(* PLC project Display.project, CODESYS V3.5 SP19 Patch 6 *)
(* stored: creationDateTime 2026-03-19T14:01:24.3469953+02:00, modificationDateTime 2026-03-19T14:01:24.3469953+02:00 *)

TYPE IdentityObject : STRUCT
  VendorId : DWORD := 0;  (* Vendor ID *)
  ProductCode : DWORD := 0;  (* Product code *)
  Revision : DWORD := 0;  (* Revision number *)
  SerialNumber : DWORD := 0;  (* Serial number for control unit *)
END_STRUCT;
END_TYPE

TYPE InitCanProtocolStates : (INIT_CANOPEN_PROTOCOLS := 1, INIT_CANOPEN_OD := 2, INIT_CANOPEN_PDO := 3, INIT_CANOPEN_OD_SAVE := 4, INIT_CANOPEN_OD_REORG := 5, INIT_CANOPEN_OD_REORG_READY := 6, INIT_INITIALIZE_OD_PARAMS := 7, INIT_INITIALIZE_OD_PARAMS_READY := 8, INIT_J1939 := 9, INIT_PROTOCOLS_DONE := 10);
END_TYPE

TYPE CAN1_TPDO_Bits : STRUCT
  Enable : BIT;  (* Bit[0] *)
  Set_BITS_Bit1 : BIT;  (* Bit[1] *)
  Set_BITS_Bit2 : BIT;  (* Bit[2] *)
  Set_BITS_Bit3 : BIT;  (* Bit[3] *)
  Set_BITS_Bit4 : BIT;  (* Bit[4] *)
  Set_BITS_Bit5 : BIT;  (* Bit[5] *)
  Set_BITS_Bit6 : BIT;  (* Bit[6] *)
  Set_BITS_Bit7 : BIT;  (* Bit[7] *)
END_STRUCT;
END_TYPE

TYPE CAN1_RPDO_RAU_Bits : STRUCT
  RAU_GPS_Init : BIT;  (* Bit[0] *)
  RAU_Bits_Bit1 : BIT;  (* Bit[1] *)
  RAU_Bits_Bit2 : BIT;  (* Bit[2] *)
  RAU_Bits_Bit3 : BIT;  (* Bit[3] *)
  RAU_Bits_Bit4 : BIT;  (* Bit[4] *)
  RAU_Bits_Bit5 : BIT;  (* Bit[5] *)
  RAU_Bits_Bit6 : BIT;  (* Bit[6] *)
  RAU_Bits_Bit7 : BIT;  (* Bit[7] *)
END_STRUCT;
END_TYPE

PROGRAM Main

                    
                      /// User code should be added to POU named as Main.
                    
                  
END_PROGRAM

PROGRAM MainInit
  VAR_OUTPUT
    o_MainInitReady : BOOL := FALSE;
  END_VAR

                    o_MainInitReady := TRUE;
                  
END_PROGRAM

(* Tool version : '8.6.9547.24640' (MultiTool build version) Xml version : '5.2' (MultiTool xml file version) Control Unit : 'Display' (Name of the unit in MultiTool) Control Unit Type : '6807' (Type of the unit in MultiTool, including the functional version) CODESYS Profile : 'CODESYS V3.5 SP19 Patch 6' (CODESYS profile that was selected in MultiTool) Device Description Version: '2.1.0.8' (Device description version that was selected in MultiTool) Export Time : '19.03.2026 14.01.24' (Date and time when exported from MultiTool) Export Path : 'C:\Codesys RPC\apps\CodesysRPC\Display' (Path where MultiTool exported) Project File : 'C:\Codesys RPC\apps\CodesysRPC\CodesysRPC.mtproject' (MultiTool project file name that was used) Libraries Path : 'C:\Codesys RPC\apps\CodesysRPC\Display\Libraries' *)
PROGRAM PLC_PRG

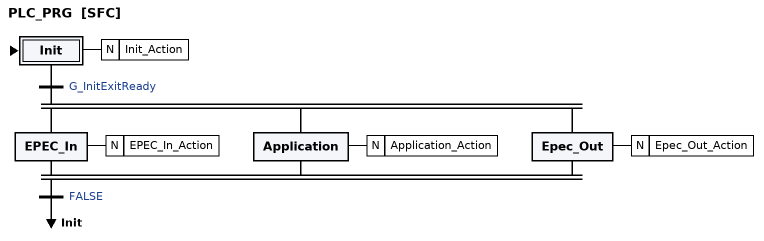
INITIAL_STEP Init:
  Init_Action(N);
END_STEP
TRANSITION FROM Init TO (EPEC_In, Application, Epec_Out)
  := G_InitExitReady;
END_TRANSITION
STEP EPEC_In:
  EPEC_In_Action(N);
END_STEP
TRANSITION FROM (EPEC_In, Application, Epec_Out) TO Init
  := FALSE;
END_TRANSITION
STEP Application:
  Application_Action(N);
END_STEP
STEP Epec_Out:
  Epec_Out_Action(N);
END_STEP

ACTION Application_Action:
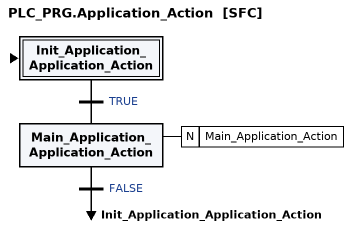
INITIAL_STEP Init_Application_Application_Action:
END_STEP
TRANSITION FROM Init_Application_Application_Action TO Main_Application_Application_Action
  := TRUE;
END_TRANSITION
STEP Main_Application_Application_Action:
  Main_Application_Action(N);
END_STEP
TRANSITION FROM Main_Application_Application_Action TO Init_Application_Application_Action
  := FALSE;
END_TRANSITION
END_ACTION

ACTION Bus_Action:
                        

G_CAN1_Channel.CheckMessages();
G_CAN2_Channel.CheckMessages();

(* Update callback data *)
IF G_CAN1_Channel.GetLatestError() <> DWORD#0 THEN
	G_CANopen_CAN1_VAR.Callback_Error := EPEC_CANopen.Errors.CallbackError;
ELSE
	G_CANopen_CAN1_VAR.Callback_Error := EPEC_CANopen.Errors.NoError;
END_IF

(* Update protocol data *)
G_CANopen_CAN1.HB_Handler.Update(
	i_Enable := TRUE,
	o_Error => G_CANopen_CAN1_VAR.HB_Error
);
G_CANopen_CAN1.NMT_Handler.Update(
	i_Enable := TRUE,
	o_Error => G_CANopen_CAN1_VAR.NMT_Error
);
G_CANopen_CAN1.SSDO_Handler.Update(
	i_Enable := TRUE,
	o_Error => G_CANopen_CAN1_VAR.SSDO_Error
);
G_CANopen_CAN1.GFC_Handler.Update(
	i_Enable := TRUE,
	o_Error => G_CANopen_CAN1_VAR.GFC_Error
);
G_CANopen_CAN1.PDO_Handler.Update(
	i_Enable := TRUE,
	o_Error => G_CANopen_CAN1_VAR.PDO_Error
);

G_CANopen_CAN1.OD_ReOrg.Update(o_Ready => , o_Error => G_CANopen_CAN1_VAR.OD_REORG_Error);

G_CANopen_CAN1.SaveODHandler.Update(i_Enable := TRUE,
	o_Ready => G_CANopen_CAN1_VAR.ODSave_OperationReady,
	o_Error => G_CANopen_CAN1_VAR.ODSave_Error);

IF G_CANopen_CAN1_VAR.HB_Error = EPEC_CANopen.Errors.NoError AND
	G_CANopen_CAN1_VAR.NMT_Error = EPEC_CANopen.Errors.NoError AND
	G_CANopen_CAN1_VAR.SSDO_Error = EPEC_CANopen.Errors.NoError AND
	G_CANopen_CAN1_VAR.GFC_Error = EPEC_CANopen.Errors.NoError AND
	G_CANopen_CAN1_VAR.PDO_Error = EPEC_CANopen.Errors.NoError AND
	G_CANopen_CAN1_VAR.OD_REORG_Error = EPEC_CANopen.Errors.NoError
THEN
	G_CANopenCan1ProtocolError := FALSE;
ELSE
	G_CANopenCan1ProtocolError := TRUE;
END_IF



(*Check for nmt reset *)
IF G_CANopen_CAN1.NMT.StateChanged THEN
	IF G_CANopen_CAN1.NMT.LastNmtCommand = EPEC_CANopen.NMTCommand.Reset OR 
	   G_CANopen_CAN1.NMT.LastNmtCommand = EPEC_CANopen.NMTCommand.ResetCommunication 
	THEN
		(* If there is NMT reset command for IEC application CANopen device,
			IEC application is started after IEC cycle in execution. *)
		G_RESET_MODULE := TRUE;
	END_IF
END_IF




                        
                      
END_ACTION

ACTION Diag_Action:
                        


(* HW diagnostic *)
    G_HWDiagnostics(
        i_SupplyVoltage  := WORD_TO_UINT(DEV_DSC_SUPPLY_Volt),
        i_SupplyVoltageHighLimit := G_SupplyVoltageHighLimit,
        i_SupplyVoltageLowLimit :=G_SupplyVoltageLowLimit,
        i_Ref5V := WORD_TO_UINT(DEV_DSC_REF_5V),
        i_Ref5VHighLimit :=  G_Ref5VHighLimit,
        i_Ref5VLowLimit := G_Ref5VLowLimit,
        i_PCBTemperature := DEV_DSC_TEMP_PCB,
        i_PCBTempHighLimit := G_TempPCBHighLimit,
        i_PCBTempLowLimit := G_TempPCBLowLimit,
        i_CPUTemperature := DEV_DSC_TEMP_CPU,
        i_CPUTempHighLimit := G_TempCPUHighLimit,
        i_CPUTempLowLimit := G_TempCPULowLimit,
        i_CycleTimeHighLimit := G_CycleTimeHighLimit,
        i_AIBiasVoltage	:= WORD_TO_UINT(DEV_DSC_AI_BIAS_Volt),
        i_RtcBackupVoltage := WORD_TO_UINT(DEV_DSC_RTC_BACKUP_Volt),
        i_Voltage12V := 0,
        i_AIBiasVoltageHighLimit := G_AIBiasVoltageHighLimit,
        i_AIBiasVoltageLowLimit := G_AIBiasVoltageLowLimit,
        i_RtcBackupVoltageLowLimit := G_RTCBackupVoltageLowLimit,
        i_Voltage12VHighLimit := 0,
        i_Voltage12VLowLimit := 0
    );

    SUPPLY_Volt := G_HWDiagnostics.o_SupplyVoltage;
    TEMP_PCB := G_HWDiagnostics.o_PCBTemperature;
    TEMP_CPU := G_HWDiagnostics.o_CPUTemperature;
    DEV_DSC_REF_OUT_5V_Enable := REF_OUT_5V_Enable;
    REF_OUT_5V_OK := (NOT DEV_DSC_REF_OUT_5V_ERROR) AND REF_OUT_5V_Enable;
	REF_5V := G_HWDiagnostics.o_Ref5V;
	AIBias_Volt := G_HWDiagnostics.o_AIBiasVoltage;
	RTCBackup_Volt := G_HWDiagnostics.o_RtcBackupVoltage;
	Voltage12V := G_HWDiagnostics.o_Voltage12V;
	ALS_Volt := DEV_DSC_ALS_Volt;

(* DO Sensing *)
	HWD_DOSensing_68xx(i_MeasuredVoltage := DEV_DSC_DO_DIAG_Volt);
	DEV_DSC_DO_DIAG_Enable := HWD_DOSensing_68xx.o_Enable;
	DEV_DSC_DO_DIAG_Selection := HWD_DOSensing_68xx.o_PinSelection;








(*########################################################*)
(*This block is created implicit. Don't add own code here.*)
(*########################################################*)

(* Diagnostics for CAN interfaces *)



(* CANopen networks management and diagnostics  *)



(* System Ok conditions *)
G_SystemOk:=NOT(G_HWDiagnostics.o_CPUTemperatureHigh) AND
		NOT(G_HWDiagnostics.o_CPUTemperatureLow) AND
		NOT(G_HWDiagnostics.o_PCBTemperatureHigh) AND
		NOT(G_HWDiagnostics.o_PCBTemperatureLow) AND
		NOT(G_HWDiagnostics.o_SupplyVoltageHigh) AND
		NOT(G_HWDiagnostics.o_SupplyVoltageLow) AND
		NOT(G_HWDiagnostics.o_CycleTimeHigh) AND
		NOT(G_HWDiagnostics.o_Ref5VHigh) AND
		NOT(G_HWDiagnostics.o_Ref5VLow) AND
		NOT(G_HWDiagnostics.o_AIBiasVoltageHigh) AND
		NOT(G_HWDiagnostics.o_AIBiasVoltageLow);

                        
                      
END_ACTION

ACTION EPEC_In_Action:
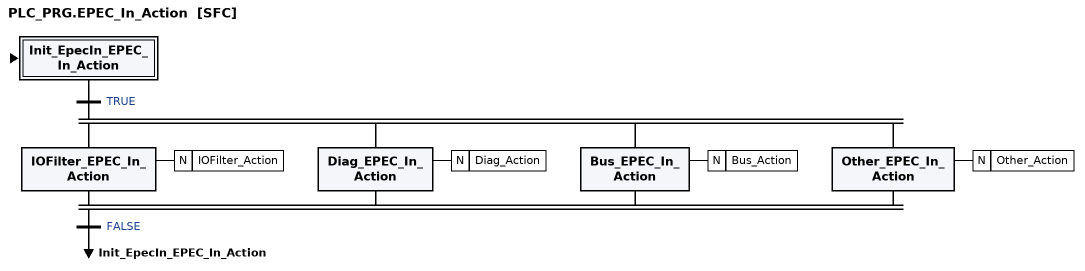
INITIAL_STEP Init_EpecIn_EPEC_In_Action:
END_STEP
TRANSITION FROM Init_EpecIn_EPEC_In_Action TO (IOFilter_EPEC_In_Action, Diag_EPEC_In_Action, Bus_EPEC_In_Action, Other_EPEC_In_Action)
  := TRUE;
END_TRANSITION
STEP IOFilter_EPEC_In_Action:
  IOFilter_Action(N);
END_STEP
TRANSITION FROM (IOFilter_EPEC_In_Action, Diag_EPEC_In_Action, Bus_EPEC_In_Action, Other_EPEC_In_Action) TO Init_EpecIn_EPEC_In_Action
  := FALSE;
END_TRANSITION
STEP Diag_EPEC_In_Action:
  Diag_Action(N);
END_STEP
STEP Bus_EPEC_In_Action:
  Bus_Action(N);
END_STEP
STEP Other_EPEC_In_Action:
  Other_Action(N);
END_STEP
END_ACTION

ACTION Epec_Out_Action:
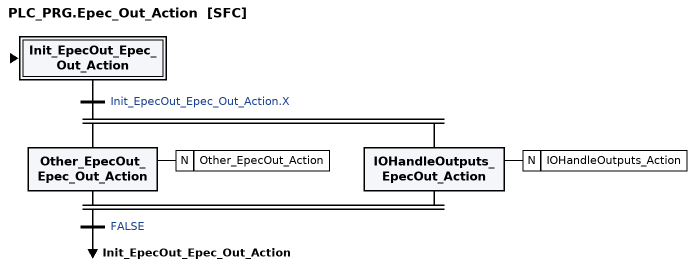
INITIAL_STEP Init_EpecOut_Epec_Out_Action:
END_STEP
TRANSITION FROM Init_EpecOut_Epec_Out_Action TO (Other_EpecOut_Epec_Out_Action, IOHandleOutputs_EpecOut_Action)
  := Init_EpecOut_Epec_Out_Action.X;
END_TRANSITION
STEP Other_EpecOut_Epec_Out_Action:
  Other_EpecOut_Action(N);
END_STEP
TRANSITION FROM (Other_EpecOut_Epec_Out_Action, IOHandleOutputs_EpecOut_Action) TO Init_EpecOut_Epec_Out_Action
  := FALSE;
END_TRANSITION
STEP IOHandleOutputs_EpecOut_Action:
  IOHandleOutputs_Action(N);
END_STEP
END_ACTION

ACTION Init_Action:
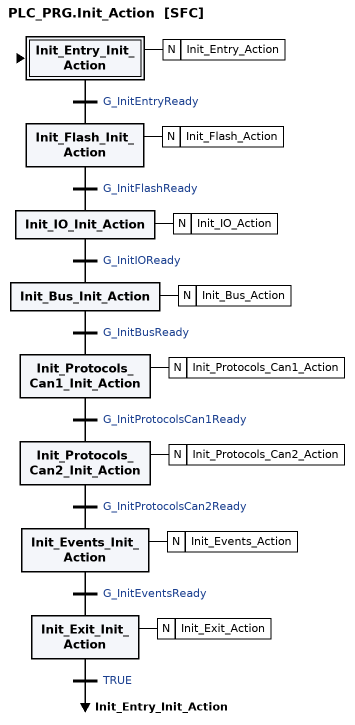
INITIAL_STEP Init_Entry_Init_Action:
  Init_Entry_Action(N);
END_STEP
TRANSITION FROM Init_Entry_Init_Action TO Init_Flash_Init_Action
  := G_InitEntryReady;
END_TRANSITION
STEP Init_Flash_Init_Action:
  Init_Flash_Action(N);
END_STEP
TRANSITION FROM Init_Flash_Init_Action TO Init_IO_Init_Action
  := G_InitFlashReady;
END_TRANSITION
STEP Init_IO_Init_Action:
  Init_IO_Action(N);
END_STEP
TRANSITION FROM Init_IO_Init_Action TO Init_Bus_Init_Action
  := G_InitIOReady;
END_TRANSITION
STEP Init_Bus_Init_Action:
  Init_Bus_Action(N);
END_STEP
TRANSITION FROM Init_Bus_Init_Action TO Init_Protocols_Can1_Init_Action
  := G_InitBusReady;
END_TRANSITION
STEP Init_Protocols_Can1_Init_Action:
  Init_Protocols_Can1_Action(N);
END_STEP
TRANSITION FROM Init_Protocols_Can1_Init_Action TO Init_Protocols_Can2_Init_Action
  := G_InitProtocolsCan1Ready;
END_TRANSITION
STEP Init_Protocols_Can2_Init_Action:
  Init_Protocols_Can2_Action(N);
END_STEP
TRANSITION FROM Init_Protocols_Can2_Init_Action TO Init_Events_Init_Action
  := G_InitProtocolsCan2Ready;
END_TRANSITION
STEP Init_Events_Init_Action:
  Init_Events_Action(N);
END_STEP
TRANSITION FROM Init_Events_Init_Action TO Init_Exit_Init_Action
  := G_InitEventsReady;
END_TRANSITION
STEP Init_Exit_Init_Action:
  Init_Exit_Action(N);
END_STEP
TRANSITION FROM Init_Exit_Init_Action TO Init_Entry_Init_Action
  := TRUE;
END_TRANSITION
END_ACTION

ACTION Init_Bus_Action:
                        (*###########################################################*)
(*This block is created implicit. Don't add own code to here.*)
(*###########################################################*)

G_CAN1_Channel.InitCAN(i_Channel:= EPEC_6000CANVXD.GVL_6000.CAN1, i_BitRate:=EPEC_CANVXD.BITRATE_250K, i_Flags:= 0);




G_InitBusReady := TRUE;

                        
                      
END_ACTION

ACTION Init_Entry_Action:
                        (*###########################################################*)
(*This block is created implicit. Don't add own code to here.*)
(*###########################################################*)

/// Call user init until flag is set on.
MainInit();
G_InitEntryReady := MainInit.o_MainInitReady;

IF TRUE = G_InitEntryReady THEN

EPEC_6000INT.GetUserFolder(i_pPath:=ADR(G_UserFolderPath),i_Length:=SIZEOF(G_UserFolderPath));


END_IF
                        
                      
END_ACTION

ACTION Init_Events_Action:
                        (*###########################################################*)
(*This block is created implicit. Don't add own code to here.*)
(*###########################################################*)
;



G_InitEventsReady:=TRUE;
                        
                      
END_ACTION

ACTION Init_Exit_Action:
                        (*###########################################################*)
(*This block is created implicit. Don't add own code to here.*)
(*###########################################################*)
;

G_NETWORK1_Parameters_CsvFile := Standard.CONCAT(STR1:=G_UserFolderPath, STR2:=G_NETWORK1_Parameters_CsvFile);
G_NETWORK1_Parameters_Count := EPEC_PAR.PARAMETERS_ReadCSV(i_Enable:=TRUE,
	i_File:=G_NETWORK1_Parameters_CsvFile,
	i_ParameterMaxCount:=G_NUMBER_OF_PARAMETERS_NETWORK1,
	i_pCSV:=0,
	i_itfExtraData:=0,
	o_CSVErrorCode=>G_NETWORK1_Parameters_ErrorCode,
	o_CSVErrorLine=>G_NETWORK1_Parameters_ErrorInLine);


G_UI.TimeSyncMethod := EPEC_6000INT.TimeSyncTypes.Manual;


G_InitExitReady:=TRUE;
                        
                      
END_ACTION

ACTION Init_Flash_Action:
                        (*###########################################################*)
(*This block is created implicit. Don't add own code to here.*)
(*###########################################################*)

G_InitFlashReady:=TRUE;
                        
                      
END_ACTION

ACTION Init_IO_Action:
                        (*###########################################################*)
(*This block is created implicit. Don't add own code to here.*)
(*###########################################################*)
;
(*IO init:*)
/// Init pin to AI mode Pin 1.5
DEV_DSC_AI_SET_mA_X1_5 := AI_SET_mA_X1_5;
DEV_DSC_AI_SET_PU_X1_5 := AI_SET_PU_X1_5;

/// Init pin to AI mode Pin 1.17
DEV_DSC_AI_SET_mA_X1_17 := AI_SET_mA_X1_17;
DEV_DSC_AI_SET_PU_X1_17 := AI_SET_PU_X1_17;


(*IO-init OK?*)
G_InitIOReady:=TRUE;
                        
                      
END_ACTION

ACTION Init_Protocols_Can1_Action:
                        (*###########################################################*)
(*This block is created implicit. Don't add own code to here.*)
(*###########################################################*)
;
CASE G_InitProtocolsCan1State OF

InitCanProtocolStates.INIT_CANOPEN_PROTOCOLS:
(*CAN1 INIT*)

G_CANopen_CAN1.Device.itfCanChannel:=G_CAN1_Channel; (*Connect device to can channel*)
G_CANopen_CAN1.Device.NodeID := BYTE#2;
G_CANopen_CAN1.NMT.NmtState:=EPEC_CANopen.NMTState.BootUp; (* Set NMT status to BOOTUP *)

(*Initialize OD's data structures*)
G_CANopen_CAN1.OD.EntryCount:=SIZEOF(G_CANopen_CAN1.ODEntrys)/SIZEOF(G_CANopen_CAN1.ODEntrys[1]); (*Max entries of given OD(CANopenDeviceODEntrys array)*)
G_CANopen_CAN1.OD.InOrder:=FALSE; (*OD isn't in order*)
G_CANopen_CAN1.OD.NextFree:=0; (*OD does not have any entries yet*)
G_CANopen_CAN1.OD.pODEntry:=ADR(G_CANopen_CAN1.ODEntrys); (*Pointer to OD array*)

(*Define NMT protocol*)
G_CANopen_CAN1.Protocols[1].Protocol:=EPEC_CANopen.ProtocolType.NMT;
G_CANopen_CAN1.Protocols[1].pData:=ADR(G_CANopen_CAN1.NMT);
G_CANopen_CAN1.Protocols[1].itfProtocol:=G_CANopen_CAN1.NMT_Handler;
G_CANopen_CAN1.Protocols[1].pError:=ADR(G_CANopen_CAN1_VAR.NMT_Error);
G_CANopen_CAN1_VAR.ProtocolAdded[1] := CANopenDeviceAddProtocol( (* Add to protocol stack *)
	i_pDevice:=ADR(G_CANopen_CAN1.Device),
	i_pProtocol:=ADR(G_CANopen_CAN1.Protocols[1]),
);

(*Initialize NMT protocol*)
IF G_CANopen_CAN1_VAR.ProtocolAdded[1] THEN
	G_CANopen_CAN1.NMT_Handler.Init(
		i_pDevice := ADR(G_CANopen_CAN1.Device),
		i_ThisIsMaster := TRUE,
		i_StartInterval :=  1000,
		i_pMonitoredNodes := ADR(G_CANopen_CAN1.MonitoredNodes),
		i_NumberOfNodes := 1,
		i_SimultaneousSlaveConfiguration := FALSE,
		i_pOdReOrg := ADR(G_CANopen_CAN1.OD_ReOrg),
		o_Error => G_CANopen_CAN1_VAR.NMT_Error
	);
ELSE
	G_CANopen_CAN1_VAR.NMT_Error := EPEC_CANopen.Errors.ProtocolDataMissing;
END_IF

(*Define OD protocol*)
G_CANopen_CAN1.Protocols[2].Protocol:=EPEC_CANopen.ProtocolType.OD;
G_CANopen_CAN1.Protocols[2].pData:=ADR(G_CANopen_CAN1.OD);
G_CANopen_CAN1.Protocols[2].pError:=ADR(G_CANopen_CAN1_VAR.OD_Error);
G_CANopen_CAN1_VAR.ProtocolAdded[2] := CANopenDeviceAddProtocol( (* Add to protocol stack *)
	i_pDevice:=ADR(G_CANopen_CAN1.Device),
	i_pProtocol:=ADR(G_CANopen_CAN1.Protocols[2]),
);
IF NOT G_CANopen_CAN1_VAR.ProtocolAdded[2] THEN
	G_CANopen_CAN1_VAR.OD_Error := EPEC_CANopen.Errors.ProtocolDataMissing;
END_IF

	(*Define HB protocol
	- Uses NMT and OD protocol data, thus need to be defined after them.
	*)
	G_CANopen_CAN1.HB.HeartBeat.PT := T#200MS; (* HB producer time *)
	G_CANopen_CAN1.HB.pHBCTimes := ADR(G_CANopen_CAN1_VAR.HBCTimes); (* HB consumer times *)

	G_CANopen_CAN1.Protocols[3].Protocol:=EPEC_CANopen.ProtocolType.HB;
	G_CANopen_CAN1.Protocols[3].pData:=ADR(G_CANopen_CAN1.HB);
	G_CANopen_CAN1.Protocols[3].itfProtocol:=G_CANopen_CAN1.HB_Handler;
	G_CANopen_CAN1.Protocols[3].pError:=ADR(G_CANopen_CAN1_VAR.HB_Error);
	G_CANopen_CAN1_VAR.ProtocolAdded[3] := CANopenDeviceAddProtocol( (* Add to protocol stack *)
		i_pDevice:=ADR(G_CANopen_CAN1.Device),
		i_pProtocol:=ADR(G_CANopen_CAN1.Protocols[3]),
	);

	(* Initialize HB protocol *)
	IF G_CANopen_CAN1_VAR.ProtocolAdded[3] THEN

		(* Add monitored nodes *)
		G_CANopen_CAN1.HB_Handler.AddCallbackToList(
			i_pDevice := ADR(G_CANopen_CAN1.Device),
			i_pCallback:=ADR(G_CANopen_CAN1.HBCallbacks[1]),
			o_Error => G_CANopen_CAN1_VAR.HB_Error
		);
		IF G_CANopen_CAN1_VAR.HB_Error = EPEC_CANopen.Errors.NoError THEN
			G_CANopen_CAN1.HB_Handler.Init(
				i_pDevice := ADR(G_CANopen_CAN1.Device),
				o_Error => G_CANopen_CAN1_VAR.HB_Error
			);
		END_IF
	ELSE
		G_CANopen_CAN1_VAR.HB_Error := EPEC_CANopen.Errors.ProtocolDataMissing;
	END_IF


(*Define SSDO protocol*)
G_CANopen_CAN1.Protocols[4].Protocol:=EPEC_CANopen.ProtocolType.SSDO;
G_CANopen_CAN1.Protocols[4].pData:=ADR(G_CANopen_CAN1.SSDO);
G_CANopen_CAN1.Protocols[4].itfProtocol:=G_CANopen_CAN1.SSDO_Handler;
G_CANopen_CAN1.Protocols[4].pError:=ADR(G_CANopen_CAN1_VAR.SSDO_Error);
G_CANopen_CAN1_VAR.ProtocolAdded[4] := CANopenDeviceAddProtocol( (* Add to protocol stack *)
	i_pDevice:=ADR(G_CANopen_CAN1.Device),
	i_pProtocol:=ADR(G_CANopen_CAN1.Protocols[4])
);
IF G_CANopen_CAN1_VAR.ProtocolAdded[4] THEN
	G_CANopen_CAN1.SSDO_Handler.Init(
		i_pDevice := ADR(G_CANopen_CAN1.Device),
		o_Error => G_CANopen_CAN1_VAR.SSDO_Error
	);
ELSE
	G_CANopen_CAN1_VAR.SSDO_Error := EPEC_CANopen.Errors.ProtocolDataMissing;
END_IF

(*Define PDO protocol*)
G_CANopen_CAN1.Protocols[5].Protocol:=EPEC_CANopen.ProtocolType.PDO;
G_CANopen_CAN1.Protocols[5].pData:=ADR(G_CANopen_CAN1.PDO);
G_CANopen_CAN1.Protocols[5].itfProtocol:=G_CANopen_CAN1.PDO_Handler;
G_CANopen_CAN1.Protocols[5].pError:=ADR(G_CANopen_CAN1_VAR.PDO_Error);
G_CANopen_CAN1_VAR.ProtocolAdded[5] := CANopenDeviceAddProtocol( (* Add to protocol stack *)
	i_pDevice:=ADR(G_CANopen_CAN1.Device),
	i_pProtocol:=ADR(G_CANopen_CAN1.Protocols[5])
);
IF G_CANopen_CAN1_VAR.ProtocolAdded[5] THEN
	G_CANopen_CAN1.PDO_Handler.Init(
		i_pDevice := ADR(G_CANopen_CAN1.Device),
		o_Error => G_CANopen_CAN1_VAR.PDO_Error
	);
ELSE
	G_CANopen_CAN1_VAR.PDO_Error := EPEC_CANopen.Errors.ProtocolDataMissing;
END_IF

(*Define GFC protocol*)
G_CANopen_CAN1.Protocols[6].Protocol:=EPEC_CANopen.ProtocolType.GFC;
G_CANopen_CAN1.Protocols[6].pData:=ADR(G_CANopen_CAN1.GFC);
G_CANopen_CAN1.Protocols[6].itfProtocol:=G_CANopen_CAN1.GFC_Handler;
G_CANopen_CAN1.Protocols[6].pError:=ADR(G_CANopen_CAN1_VAR.GFC_Error);
G_CANopen_CAN1_VAR.ProtocolAdded[6] := CANopenDeviceAddProtocol(  (* Add to protocol stack *)
	i_pDevice:=ADR(G_CANopen_CAN1.Device),
	i_pProtocol:=ADR(G_CANopen_CAN1.Protocols[6])
);
IF G_CANopen_CAN1_VAR.ProtocolAdded[6] THEN
	G_CANopen_CAN1.GFC_Handler.Init(
		i_pDevice := ADR(G_CANopen_CAN1.Device),
		i_pStatus:=ADR(G_CANopen_CAN1_VAR.GFC_Status),
		o_Error => G_CANopen_CAN1_VAR.GFC_Error
	);
ELSE
	G_CANopen_CAN1_VAR.GFC_Error := EPEC_CANopen.Errors.ProtocolDataMissing;
END_IF

(* Init CSDO instance array for bus *)
EPEC_CANopen.CANopenSDOManager.Init(
	i_pDevice:=ADR(G_CANopen_CAN1.Device),
	i_pCsdoArrayStart:=ADR(G_CANopen_CAN1.CSDOS),
	i_CsdoArraySize:=SIZEOF(G_CANopen_CAN1.CSDOS)/SIZEOF(G_CANopen_CAN1.CSDOS[1]),
	o_Error=>G_CANopen_CAN1_VAR.CSDO_Error
);





G_InitProtocolsCan1State := InitCanProtocolStates.INIT_CANOPEN_OD;

InitCanProtocolStates.INIT_CANOPEN_OD:

(*16#0001..16#0009 Default types *)
G_CANopen_CAN1_VAR.OD_Error := EPEC_CANopen.CANopenODAddDefautTypes(
	i_pOD:= ADR(G_CANopen_CAN1.OD)
);

	(* 16#1000 Information about the device type *)
	IF G_CANopen_CAN1_VAR.OD_Error = EPEC_CANopen.Errors.NoError THEN
		G_CANopen_CAN1_VAR.OD_Error := CANopenODAddLine(
			i_pOD := ADR(G_CANopen_CAN1.OD),(*Address of Object dictionary where index will be added*)
			i_Index := G_CANOPEN_ODINDEX_DEVICE_TYPE,
			i_ObjectCode := EPEC_CANopen.ObjectCode.OD_VAR,(*Type of index*)
			i_NumOfSubids := USINT#0,(*Number of subindexes*)
			i_TypeSpec := EPEC_CANopen.DataType.Deftype_UNSIGNED32,(*Index datatype, either user defined or standard CiA 301*)
			i_ObjectAccess := G_CANOPEN_OD_ACCESS_NOWRITE OR G_CANOPEN_OD_ACCESS_SUB0NOWRITE,
			i_Sub0data := USINT#0,(*Value of subindex0 in array or (def)struct*)
			i_pIndexData := ADR(G_CAN1_VAR.DeviceType_Device1),
			i_itfSDOHandler := DWORD#0
		);
	END_IF

	(* 16#1001 Error information *)
	IF G_CANopen_CAN1_VAR.OD_Error = EPEC_CANopen.Errors.NoError THEN
		G_CANopen_CAN1_VAR.OD_Error := CANopenODAddLine(
			i_pOD := ADR(G_CANopen_CAN1.OD),(*Address of Object dictionary where index will be added*)
			i_Index := G_CANOPEN_ODINDEX_ERROR_REGISTER,
			i_ObjectCode := EPEC_CANopen.ObjectCode.OD_VAR,(*Type of index*)
			i_NumOfSubids := USINT#0,(*Number of subindexes*)
			i_TypeSpec := EPEC_CANopen.DataType.Deftype_UNSIGNED8,(*Index datatype, either user defined or standard CiA 301*)
			i_ObjectAccess := G_CANOPEN_OD_ACCESS_NOWRITE OR G_CANOPEN_OD_ACCESS_SUB0NOWRITE,
			i_Sub0data := USINT#0,(*Value of subindex0 in array or (def)struct*)
			i_pIndexData := ADR(G_CAN1_VAR.ErrorReg_Device1),
			i_itfSDOHandler := DWORD#0
		);
	END_IF

	(* 16#1008 Manufacturer device name *)
	IF G_CANopen_CAN1_VAR.OD_Error = EPEC_CANopen.Errors.NoError THEN
		G_CANopen_CAN1_VAR.OD_Error := CANopenODAddLine(
			i_pOD := ADR(G_CANopen_CAN1.OD),(*Address of Object dictionary where index will be added*)
			i_Index := G_CANOPEN_ODINDEX_MF_DEVICE_NAME,
			i_ObjectCode := EPEC_CANopen.ObjectCode.OD_VAR,(*Type of index*)
			i_NumOfSubids := USINT#0,(*Number of subindexes*)
			i_TypeSpec := EPEC_CANopen.DataType.Deftype_STRING,(*Index datatype, either user defined or standard CiA 301*)
			i_ObjectAccess := G_CANOPEN_OD_ACCESS_NOWRITE OR G_CANOPEN_OD_ACCESS_SUB0NOWRITE,
			i_Sub0data := USINT#0,(*Value of subindex0 in array or (def)struct*)
			i_pIndexData := ADR(G_SystemInfo.DeviceName),
			i_itfSDOHandler := DWORD#0
		);
	END_IF

	(* 16#100A Manufacturer software version *)
	IF G_CANopen_CAN1_VAR.OD_Error = EPEC_CANopen.Errors.NoError THEN
		G_CANopen_CAN1_VAR.OD_Error := CANopenODAddLine(
			i_pOD := ADR(G_CANopen_CAN1.OD),(*Address of Object dictionary where index will be added*)
			i_Index := G_CANOPEN_ODINDEX_MF_SW_VERSION,
			i_ObjectCode := EPEC_CANopen.ObjectCode.OD_VAR,(*Type of index*)
			i_NumOfSubids := USINT#0,(*Number of subindexes*)
			i_TypeSpec := EPEC_CANopen.DataType.Deftype_STRING,(*Index datatype, either user defined or standard CiA 301*)
			i_ObjectAccess := G_CANOPEN_OD_ACCESS_NOWRITE OR G_CANOPEN_OD_ACCESS_SUB0NOWRITE,
			i_Sub0data := USINT#0,(*Value of subindex0 in array or (def)struct*)
			i_pIndexData := ADR(G_SystemInfo.SWVersion),
			i_itfSDOHandler := DWORD#0
		);
	END_IF

	(* 16#1018   Vendor ID *)
	IF G_CANopen_CAN1_VAR.OD_Error = EPEC_CANopen.Errors.NoError THEN
		G_CANopen_CAN1_VAR.OD_Error := CANopenODAddLine(
			i_pOD := ADR(G_CANopen_CAN1.OD),(*Address of Object dictionary where index will be added*)
			i_Index := G_CANOPEN_ODINDEX_IDENTITY_OBJECT,
			i_ObjectCode := EPEC_CANopen.ObjectCode.OD_ARRAY, (*Type of index*)
			i_NumOfSubids := USINT#4,(*Number of subindexes*)
			i_TypeSpec := EPEC_CANopen.DataType.Deftype_UNSIGNED32,(*Index of 16-bit deftype*)
			i_ObjectAccess := G_CANOPEN_OD_ACCESS_NOWRITE OR G_CANOPEN_OD_ACCESS_SUB0NOWRITE,
			i_Sub0data := USINT#4,(*Value of subindex0 in array or (def)struct*)
			i_pIndexData := ADR(G_SystemInfo.Identity),
			i_itfSDOHandler := DWORD#0
		);
	END_IF
	(* 16#2030   CodesysVersion *)
	IF G_CANopen_CAN1_VAR.OD_Error = EPEC_CANopen.Errors.NoError THEN
		G_CANopen_CAN1_VAR.OD_Error := CANopenODAddLine(
			i_pOD := ADR(G_CANopen_CAN1.OD),(*Address of Object dictionary where index will be added*)
			i_Index := 16#2030,
			i_ObjectCode := EPEC_CANopen.ObjectCode.OD_ARRAY, (*Type of index*)
			i_NumOfSubids := USINT#1,(*Number of subindexes*)
			i_TypeSpec := EPEC_CANopen.DataType.Deftype_UNSIGNED32,(*Index of 16-bit deftype*)
			i_ObjectAccess := G_CANOPEN_OD_ACCESS_READWRITE OR G_CANOPEN_OD_ACCESS_SUB0NOWRITE,
			i_Sub0data := USINT#1,(*Value of subindex0 in array or (def)struct*)
			i_pIndexData := ADR(G_SystemInfo.ToolsVersion),
			i_itfSDOHandler := DWORD#0
		);
	END_IF

	(* 16#2128 PDO Dummy Variable Index *)
	IF G_CANopen_CAN1_VAR.OD_Error = EPEC_CANopen.Errors.NoError THEN
		G_CANopen_CAN1_VAR.OD_Error := CANopenODAddLine(
			i_pOD := ADR(G_CANopen_CAN1.OD),(*Address of Object dictionary where index will be added*)
			i_Index := 16#2128,
			i_ObjectCode := EPEC_CANopen.ObjectCode.OD_VAR,(*Type of index*)
			i_NumOfSubids := USINT#0,(*Number of subindexes*)
			i_TypeSpec := EPEC_CANopen.DataType.Deftype_UNSIGNED8,(*Index datatype, either user defined or standard CiA 301*)
			i_ObjectAccess := G_CANOPEN_OD_ACCESS_READWRITE,
			i_Sub0data := USINT#0,(*Value of subindex0 in array or (def)struct*)
			i_pIndexData := ADR(G_CAN1_VAR.CAN1_TPDO_DUMMY),
			i_itfSDOHandler := DWORD#0
		);
	END_IF

	(* 16#2129 PDO Dummy Variable Index *)
	IF G_CANopen_CAN1_VAR.OD_Error = EPEC_CANopen.Errors.NoError THEN
		G_CANopen_CAN1_VAR.OD_Error := CANopenODAddLine(
			i_pOD := ADR(G_CANopen_CAN1.OD),(*Address of Object dictionary where index will be added*)
			i_Index := 16#2129,
			i_ObjectCode := EPEC_CANopen.ObjectCode.OD_VAR,(*Type of index*)
			i_NumOfSubids := USINT#0,(*Number of subindexes*)
			i_TypeSpec := EPEC_CANopen.DataType.Deftype_UNSIGNED8,(*Index datatype, either user defined or standard CiA 301*)
			i_ObjectAccess := G_CANOPEN_OD_ACCESS_READWRITE,
			i_Sub0data := USINT#0,(*Value of subindex0 in array or (def)struct*)
			i_pIndexData := ADR(G_CAN1_VAR.CAN1_RPDO_DUMMY),
			i_itfSDOHandler := DWORD#0
		);
	END_IF

	(* 16#2130   Application version *)
	IF G_CANopen_CAN1_VAR.OD_Error = EPEC_CANopen.Errors.NoError THEN
		G_CANopen_CAN1_VAR.OD_Error := CANopenODAddLine(
			i_pOD := ADR(G_CANopen_CAN1.OD),(*Address of Object dictionary where index will be added*)
			i_Index := 16#2130,
			i_ObjectCode := EPEC_CANopen.ObjectCode.OD_ARRAY, (*Type of index*)
			i_NumOfSubids := USINT#10,(*Number of subindexes*)
			i_TypeSpec := EPEC_CANopen.DataType.Deftype_STRING,(*Index of 16-bit deftype*)
			i_ObjectAccess := G_CANOPEN_OD_ACCESS_NOWRITE OR G_CANOPEN_OD_ACCESS_SUB0NOWRITE,
			i_Sub0data := USINT#10,(*Value of subindex0 in array or (def)struct*)
			i_pIndexData := ADR(G_SystemInfo.SoftwareInformation),
			i_itfSDOHandler := DWORD#0
		);
	END_IF

	(* 16#2131 Parameter CSV unique ID *)
	IF G_CANopen_CAN1_VAR.OD_Error = EPEC_CANopen.Errors.NoError THEN
		G_CANopen_CAN1_VAR.OD_Error := CANopenODAddLine(
			i_pOD := ADR(G_CANopen_CAN1.OD),(*Address of Object dictionary where index will be added*)
			i_Index := 16#2131,
			i_ObjectCode := EPEC_CANopen.ObjectCode.OD_VAR,(*Type of index*)
			i_NumOfSubids := USINT#0,(*Number of subindexes*)
			i_TypeSpec := EPEC_CANopen.DataType.Deftype_UNSIGNED16,(*Index datatype, either user defined or standard CiA 301*)
			i_ObjectAccess := G_CANOPEN_OD_ACCESS_NOWRITE OR G_CANOPEN_OD_ACCESS_SUB0NOWRITE,
			i_Sub0data := USINT#0,(*Value of subindex0 in array or (def)struct*)
			i_pIndexData := ADR(G_CAN1_VAR.Parameter_CSV_unique_ID1),
			i_itfSDOHandler := DWORD#0
		);
	END_IF

	(* 16#2140   MAC address byte 1 *)
	IF G_CANopen_CAN1_VAR.OD_Error = EPEC_CANopen.Errors.NoError THEN
		G_CANopen_CAN1_VAR.OD_Error := CANopenODAddLine(
			i_pOD := ADR(G_CANopen_CAN1.OD),(*Address of Object dictionary where index will be added*)
			i_Index := 16#2140,
			i_ObjectCode := EPEC_CANopen.ObjectCode.OD_ARRAY, (*Type of index*)
			i_NumOfSubids := USINT#6,(*Number of subindexes*)
			i_TypeSpec := EPEC_CANopen.DataType.Deftype_UNSIGNED8,(*Index of 16-bit deftype*)
			i_ObjectAccess := G_CANOPEN_OD_ACCESS_NOWRITE OR G_CANOPEN_OD_ACCESS_SUB0NOWRITE,
			i_Sub0data := USINT#6,(*Value of subindex0 in array or (def)struct*)
			i_pIndexData := ADR(G_SystemInfo.MACAddress),
			i_itfSDOHandler := DWORD#0
		);
	END_IF

	(* 16#2141   Ethernet enabled/disabled *)
	IF G_CANopen_CAN1_VAR.OD_Error = EPEC_CANopen.Errors.NoError THEN
		G_CANopen_CAN1_VAR.OD_Error := CANopenODAddLine(
			i_pOD := ADR(G_CANopen_CAN1.OD),(*Address of Object dictionary where index will be added*)
			i_Index := 16#2141,
			i_ObjectCode := EPEC_CANopen.ObjectCode.OD_ARRAY, (*Type of index*)
			i_NumOfSubids := USINT#50,(*Number of subindexes*)
			i_TypeSpec := EPEC_CANopen.DataType.Deftype_UNSIGNED8,(*Index of 16-bit deftype*)
			i_ObjectAccess := G_CANOPEN_OD_ACCESS_READWRITE OR G_CANOPEN_OD_ACCESS_SUB0NOWRITE,
			i_Sub0data := USINT#50,(*Value of subindex0 in array or (def)struct*)
			i_pIndexData := ADR(G_SystemInfo.EthernetConfiguration),
			i_itfSDOHandler := DWORD#0
		);
	END_IF

	(* 16#2150   Codesys communication enabled *)
	IF G_CANopen_CAN1_VAR.OD_Error = EPEC_CANopen.Errors.NoError THEN
		G_CANopen_CAN1_VAR.OD_Error := CANopenODAddLine(
			i_pOD := ADR(G_CANopen_CAN1.OD),(*Address of Object dictionary where index will be added*)
			i_Index := 16#2150,
			i_ObjectCode := EPEC_CANopen.ObjectCode.OD_ARRAY, (*Type of index*)
			i_NumOfSubids := USINT#10,(*Number of subindexes*)
			i_TypeSpec := EPEC_CANopen.DataType.Deftype_UNSIGNED16,(*Index of 16-bit deftype*)
			i_ObjectAccess := G_CANOPEN_OD_ACCESS_READWRITE OR G_CANOPEN_OD_ACCESS_SUB0NOWRITE,
			i_Sub0data := USINT#10,(*Value of subindex0 in array or (def)struct*)
			i_pIndexData := ADR(G_SystemInfo.CAN1_Comms),
			i_itfSDOHandler := DWORD#0
		);
	END_IF

	(* 16#2151   Codesys communication enabled *)
	IF G_CANopen_CAN1_VAR.OD_Error = EPEC_CANopen.Errors.NoError THEN
		G_CANopen_CAN1_VAR.OD_Error := CANopenODAddLine(
			i_pOD := ADR(G_CANopen_CAN1.OD),(*Address of Object dictionary where index will be added*)
			i_Index := 16#2151,
			i_ObjectCode := EPEC_CANopen.ObjectCode.OD_ARRAY, (*Type of index*)
			i_NumOfSubids := USINT#10,(*Number of subindexes*)
			i_TypeSpec := EPEC_CANopen.DataType.Deftype_UNSIGNED16,(*Index of 16-bit deftype*)
			i_ObjectAccess := G_CANOPEN_OD_ACCESS_READWRITE OR G_CANOPEN_OD_ACCESS_SUB0NOWRITE,
			i_Sub0data := USINT#10,(*Value of subindex0 in array or (def)struct*)
			i_pIndexData := ADR(G_SystemInfo.CAN2_Comms),
			i_itfSDOHandler := DWORD#0
		);
	END_IF

	(* 16#21EE Authentication status for non-safety parameter editing *)
	IF G_CANopen_CAN1_VAR.OD_Error = EPEC_CANopen.Errors.NoError THEN
		G_CANopen_CAN1_VAR.OD_Error := CANopenODAddLine(
			i_pOD := ADR(G_CANopen_CAN1.OD),(*Address of Object dictionary where index will be added*)
			i_Index := 16#21EE,
			i_ObjectCode := EPEC_CANopen.ObjectCode.OD_VAR,(*Type of index*)
			i_NumOfSubids := USINT#0,(*Number of subindexes*)
			i_TypeSpec := EPEC_CANopen.DataType.Deftype_UNSIGNED8,(*Index datatype, either user defined or standard CiA 301*)
			i_ObjectAccess := G_CANOPEN_OD_ACCESS_NOWRITE OR G_CANOPEN_OD_ACCESS_SUB0NOWRITE,
			i_Sub0data := USINT#0,(*Value of subindex0 in array or (def)struct*)
			i_pIndexData := ADR(G_CAN1_VAR.NonSafetyParameterAuthenticationStatus),
			i_itfSDOHandler := DWORD#0
		);
	END_IF

	(* 16#21EF Non-safety parameter password *)
	IF G_CANopen_CAN1_VAR.OD_Error = EPEC_CANopen.Errors.NoError THEN
		G_CANopen_CAN1_VAR.OD_Error := CANopenODAddLine(
			i_pOD := ADR(G_CANopen_CAN1.OD),(*Address of Object dictionary where index will be added*)
			i_Index := 16#21EF,
			i_ObjectCode := EPEC_CANopen.ObjectCode.OD_VAR,(*Type of index*)
			i_NumOfSubids := USINT#0,(*Number of subindexes*)
			i_TypeSpec := EPEC_CANopen.DataType.Deftype_STRING,(*Index datatype, either user defined or standard CiA 301*)
			i_ObjectAccess := G_CANOPEN_OD_ACCESS_SUB0NOREAD OR G_CANOPEN_OD_ACCESS_NOREAD,
			i_Sub0data := USINT#0,(*Value of subindex0 in array or (def)struct*)
			i_pIndexData := ADR(G_CAN1_VAR.NonSafetyParameterPassword),
			i_itfSDOHandler := DWORD#0
		);
	END_IF

	(* 16#5FB7 Automatically created REAL variables *)
	IF G_CANopen_CAN1_VAR.OD_Error = EPEC_CANopen.Errors.NoError THEN
		G_CANopen_CAN1_VAR.OD_Error := CANopenODAddLine(
			i_pOD := ADR(G_CANopen_CAN1.OD),(*Address of Object dictionary where index will be added*)
			i_Index := 16#5FB7,
			i_ObjectCode := EPEC_CANopen.ObjectCode.OD_ARRAY,(*Type of index*)
			i_NumOfSubids := USINT#6,(*Number of subindexes*)
			i_TypeSpec := EPEC_CANopen.DataType.Deftype_REAL32,(*Index datatype, either user defined or standard CiA 301*)
			i_ObjectAccess := G_CANOPEN_OD_ACCESS_READWRITE OR G_CANOPEN_OD_ACCESS_SUB0NOWRITE OR G_CANOPEN_OD_ACCESS_PDOMAP,
			i_Sub0data := USINT#6,(*Value of subindex0 in array or (def)struct*)
			i_pIndexData := ADR(G_CAN1_RPDO.RAU_GPS_altitude),
			i_itfSDOHandler := DWORD#0
		);
	END_IF

	(* 16#5FD7 Automatically created DWORD variables *)
	IF G_CANopen_CAN1_VAR.OD_Error = EPEC_CANopen.Errors.NoError THEN
		G_CANopen_CAN1_VAR.OD_Error := CANopenODAddLine(
			i_pOD := ADR(G_CANopen_CAN1.OD),(*Address of Object dictionary where index will be added*)
			i_Index := 16#5FD7,
			i_ObjectCode := EPEC_CANopen.ObjectCode.OD_ARRAY,(*Type of index*)
			i_NumOfSubids := USINT#3,(*Number of subindexes*)
			i_TypeSpec := EPEC_CANopen.DataType.Deftype_UNSIGNED32,(*Index datatype, either user defined or standard CiA 301*)
			i_ObjectAccess := G_CANOPEN_OD_ACCESS_READWRITE OR G_CANOPEN_OD_ACCESS_SUB0NOWRITE OR G_CANOPEN_OD_ACCESS_PDOMAP,
			i_Sub0data := USINT#3,(*Value of subindex0 in array or (def)struct*)
			i_pIndexData := ADR(G_CAN1_TPDO.PT100),
			i_itfSDOHandler := DWORD#0
		);
	END_IF

	(* 16#5FFF Automatically created BYTE variables *)
	IF G_CANopen_CAN1_VAR.OD_Error = EPEC_CANopen.Errors.NoError THEN
		G_CANopen_CAN1_VAR.OD_Error := CANopenODAddLine(
			i_pOD := ADR(G_CANopen_CAN1.OD),(*Address of Object dictionary where index will be added*)
			i_Index := 16#5FFF,
			i_ObjectCode := EPEC_CANopen.ObjectCode.OD_ARRAY,(*Type of index*)
			i_NumOfSubids := USINT#2,(*Number of subindexes*)
			i_TypeSpec := EPEC_CANopen.DataType.Deftype_UNSIGNED8,(*Index datatype, either user defined or standard CiA 301*)
			i_ObjectAccess := G_CANOPEN_OD_ACCESS_READWRITE OR G_CANOPEN_OD_ACCESS_SUB0NOWRITE OR G_CANOPEN_OD_ACCESS_PDOMAP,
			i_Sub0data := USINT#2,(*Value of subindex0 in array or (def)struct*)
			i_pIndexData := ADR(G_CAN1_TPDO.Bits),
			i_itfSDOHandler := DWORD#0
		);
	END_IF



G_InitProtocolsCan1State := InitCanProtocolStates.INIT_CANOPEN_PDO;

InitCanProtocolStates.INIT_CANOPEN_PDO:

	(* Init PDOs *)
	(* TPDO1 *)
	IF G_CANopen_CAN1_VAR.PDO_Error = EPEC_CANopen.Errors.NoError THEN
		G_CANopen_CAN1.PDOS[1].Init(
			i_pDevice:= ADR(G_CANopen_CAN1.Device),
			i_PDONumber := WORD#1,
			i_PDOType := EPEC_CANopen.PDOType.TransmitPDO,
			i_COB_ID := G_CANopen_CAN1.Device.NodeID + 16#180,
			i_TransmissionType := 16#FF,
			i_InhibitTime := 100,
			i_EventTime := 300,
			i_Mapping := G_CANopen_CAN1_Mappings.PDO1_Mappings,
			i_Mappings := 1,
			o_Error => G_CANopen_CAN1_VAR.PDO_Error
			);
	END_IF

	(* TPDO2 *)
	IF G_CANopen_CAN1_VAR.PDO_Error = EPEC_CANopen.Errors.NoError THEN
		G_CANopen_CAN1.PDOS[2].Init(
			i_pDevice:= ADR(G_CANopen_CAN1.Device),
			i_PDONumber := WORD#2,
			i_PDOType := EPEC_CANopen.PDOType.TransmitPDO,
			i_COB_ID := G_CANopen_CAN1.Device.NodeID + 16#280,
			i_TransmissionType := 16#FF,
			i_InhibitTime := 100,
			i_EventTime := 300,
			i_Mapping := G_CANopen_CAN1_Mappings.PDO2_Mappings,
			i_Mappings := 2,
			o_Error => G_CANopen_CAN1_VAR.PDO_Error
			);
	END_IF

	(* RAU_TPDO1 *)
	IF G_CANopen_CAN1_VAR.PDO_Error = EPEC_CANopen.Errors.NoError THEN
		G_CANopen_CAN1.PDOS[3].Init(
			i_pDevice:= ADR(G_CANopen_CAN1.Device),
			i_PDONumber := WORD#1,
			i_PDOType := EPEC_CANopen.PDOType.ReceivePDO,
			i_COB_ID := 16#181,
			i_TransmissionType := 16#FF,
			i_InhibitTime := 100,
			i_EventTime := 0,
			i_Mapping := G_CANopen_CAN1_Mappings.PDO3_Mappings,
			i_Mappings := 2,
			o_Error => G_CANopen_CAN1_VAR.PDO_Error
		);
	END_IF

	(* RAU_TPDO2 *)
	IF G_CANopen_CAN1_VAR.PDO_Error = EPEC_CANopen.Errors.NoError THEN
		G_CANopen_CAN1.PDOS[4].Init(
			i_pDevice:= ADR(G_CANopen_CAN1.Device),
			i_PDONumber := WORD#2,
			i_PDOType := EPEC_CANopen.PDOType.ReceivePDO,
			i_COB_ID := 16#281,
			i_TransmissionType := 16#FF,
			i_InhibitTime := 100,
			i_EventTime := 0,
			i_Mapping := G_CANopen_CAN1_Mappings.PDO4_Mappings,
			i_Mappings := 2,
			o_Error => G_CANopen_CAN1_VAR.PDO_Error
		);
	END_IF

	(* RAU_TPDO3 *)
	IF G_CANopen_CAN1_VAR.PDO_Error = EPEC_CANopen.Errors.NoError THEN
		G_CANopen_CAN1.PDOS[5].Init(
			i_pDevice:= ADR(G_CANopen_CAN1.Device),
			i_PDONumber := WORD#3,
			i_PDOType := EPEC_CANopen.PDOType.ReceivePDO,
			i_COB_ID := 16#381,
			i_TransmissionType := 16#FF,
			i_InhibitTime := 100,
			i_EventTime := 0,
			i_Mapping := G_CANopen_CAN1_Mappings.PDO5_Mappings,
			i_Mappings := 2,
			o_Error => G_CANopen_CAN1_VAR.PDO_Error
		);
	END_IF

	(* RAU_TPDO4 *)
	IF G_CANopen_CAN1_VAR.PDO_Error = EPEC_CANopen.Errors.NoError THEN
		G_CANopen_CAN1.PDOS[6].Init(
			i_pDevice:= ADR(G_CANopen_CAN1.Device),
			i_PDONumber := WORD#4,
			i_PDOType := EPEC_CANopen.PDOType.ReceivePDO,
			i_COB_ID := 16#481,
			i_TransmissionType := 16#FF,
			i_InhibitTime := 100,
			i_EventTime := 0,
			i_Mapping := G_CANopen_CAN1_Mappings.PDO6_Mappings,
			i_Mappings := 2,
			o_Error => G_CANopen_CAN1_VAR.PDO_Error
		);
	END_IF

	IF G_CANopen_CAN1_VAR.PDO_Error = EPEC_CANopen.Errors.NoError THEN
		G_CANopen_CAN1.PDO.pPDO:=ADR(G_CANopen_CAN1.PDOS);
		G_CANopen_CAN1.PDO.Count:=6; (* Amount of PDOS *)
	END_IF



G_InitProtocolsCan1State := InitCanProtocolStates.INIT_CANOPEN_OD_SAVE;

InitCanProtocolStates.INIT_CANOPEN_OD_SAVE:

(*Initialize OD save*)
G_CANopen_CAN1.SaveSubData1010h.pSaveSigns := ADR(G_CANopen_CAN1_VAR.SaveSigns1010[0]);
G_CANopen_CAN1.SaveSubData1010h.NumOfEntrys := 4;
G_CANopen_CAN1.SaveSubData1010h.pSaveIndexData := ADR(G_CANopen_CAN1.SaveData[0]);
G_CANopen_CAN1.SaveData[3].itfSaveAll := G_CANopen_CAN1.SaveAll;
G_CANopen_CAN1.SaveData[3].itfDeleteAll := G_CANopen_CAN1.DeleteAll;
G_CANopen_CAN1.OD.pAdditionalData := ADR(G_CANopen_CAN1.SaveSubData1010h);

IF G_CANopen_CAN1_VAR.OD_Error = EPEC_CANopen.Errors.NoError THEN
	G_CANopen_CAN1.SaveODHandler.Init(
		i_pOD:=ADR(G_CANopen_CAN1.OD),
		i_pSaveAll:= ADR(G_CANopen_CAN1.SaveAll),
		i_pDeleteAll:= ADR(G_CANopen_CAN1.DeleteAll),
		i_pParamHandler:=ADR(G_Common.ParHandler),
		i_NumOfParamsPerCycle:= 50,
		o_Error => G_CANopen_CAN1_VAR.ODSave_Error);
END_IF

G_CANopen_CAN1.OD_ReOrg.Init(i_pOD := ADR(G_CANopen_CAN1.OD), i_NumOfODIndexPerCycle := 50);
G_CANopen_CAN1.OD_ReOrg.Start();

G_InitProtocolsCan1State := InitCanProtocolStates.INIT_CANOPEN_OD_REORG;

InitCanProtocolStates.INIT_CANOPEN_OD_REORG:

G_CANopen_CAN1.OD_ReOrg.Update(o_Ready => G_CANopen_CAN1_VAR.OdReOrgReady, o_Error => G_CANopen_CAN1_VAR.OD_REORG_Error);

IF G_CANopen_CAN1_VAR.OdReOrgReady THEN
	(* Check all protocol init status flags *)
	IF G_CANopen_CAN1_VAR.NMT_Error = EPEC_CANopen.Errors.NoError AND
		G_CANopen_CAN1_VAR.SSDO_Error = EPEC_CANopen.Errors.NoError AND
		G_CANopen_CAN1_VAR.OD_Error = EPEC_CANopen.Errors.NoError AND
		G_CANopen_CAN1_VAR.HB_Error = EPEC_CANopen.Errors.NoError AND
		G_CANopen_CAN1_VAR.CSDO_Error = EPEC_CANopen.Errors.NoError AND
		G_CANopen_CAN1_VAR.GFC_Error = EPEC_CANopen.Errors.NoError AND
		G_CANopen_CAN1_VAR.PDO_Error = EPEC_CANopen.Errors.NoError AND
		G_CANopen_CAN1_VAR.OD_REORG_Error = EPEC_CANopen.Errors.NoError
	THEN
		G_InitCANopenCan1Error := FALSE; (* No errors in protocol inits *)
	ELSE
		G_InitCANopenCan1Error := TRUE;
	END_IF
	G_InitProtocolsCan1State := InitCanProtocolStates.INIT_CANOPEN_OD_REORG_READY;
END_IF

InitCanProtocolStates.INIT_CANOPEN_OD_REORG_READY:
	G_InitProtocolsCan1State := INIT_INITIALIZE_OD_PARAMS;

INIT_INITIALIZE_OD_PARAMS:
	G_CANopen_CAN1.SaveODHandler.InitializeODParams(i_Enable:=TRUE,
		o_Ready=>G_CANopen_CAN1_VAR.ODParametersInitialized,
		o_Error=>G_CANopen_CAN1_VAR.ODSave_Error);

	IF G_CANopen_CAN1_VAR.ODParametersInitialized THEN
		G_InitProtocolsCan1State := InitCanProtocolStates.INIT_INITIALIZE_OD_PARAMS_READY;
	END_IF

INIT_INITIALIZE_OD_PARAMS_READY:


G_InitProtocolsCan1State := InitCanProtocolStates.INIT_J1939;

InitCanProtocolStates.INIT_J1939:



G_InitProtocolsCan1State := InitCanProtocolStates.INIT_PROTOCOLS_DONE;

InitCanProtocolStates.INIT_PROTOCOLS_DONE:
G_InitProtocolsCan1Ready := TRUE;

END_CASE
                        
                      
END_ACTION

ACTION Init_Protocols_Can2_Action:
                        (*###########################################################*)
(*This block is created implicit. Don't add own code to here.*)
(*###########################################################*)
;
CASE G_InitProtocolsCan2State OF

InitCanProtocolStates.INIT_CANOPEN_PROTOCOLS:
(*CAN2 INIT*)





G_InitProtocolsCan2State := InitCanProtocolStates.INIT_CANOPEN_OD;

InitCanProtocolStates.INIT_CANOPEN_OD:



G_InitProtocolsCan2State := InitCanProtocolStates.INIT_CANOPEN_PDO;

InitCanProtocolStates.INIT_CANOPEN_PDO:



G_InitProtocolsCan2State := InitCanProtocolStates.INIT_CANOPEN_OD_SAVE;

InitCanProtocolStates.INIT_CANOPEN_OD_SAVE:



G_InitProtocolsCan2State := InitCanProtocolStates.INIT_J1939;

InitCanProtocolStates.INIT_J1939:



G_InitProtocolsCan2State := InitCanProtocolStates.INIT_PROTOCOLS_DONE;

InitCanProtocolStates.INIT_PROTOCOLS_DONE:
G_InitProtocolsCan2Ready := TRUE;

END_CASE
                        
                      
END_ACTION

ACTION IOFilter_Action:
                        ;

/// Handle AI channel Pin 1.5
DEV_DSC_AI_SET_mA_X1_5 := AI_SET_mA_X1_5;
DEV_DSC_AI_SET_PU_X1_5 := AI_SET_PU_X1_5;
AI_X1_5 := DEV_DSC_AI_RAW_X1_5;
AI_PU_X1_5 := DEV_DSC_AI_PU_X1_5;


/// KL15 Pin 1.6
KL15_X1_6 := DEV_DSC_KL15;



/// Handle AI channel Pin 1.17
DEV_DSC_AI_SET_mA_X1_17 := AI_SET_mA_X1_17;
DEV_DSC_AI_SET_PU_X1_17 := AI_SET_PU_X1_17;
AI_X1_17 := DEV_DSC_AI_RAW_X1_17;
AI_PU_X1_17 := DEV_DSC_AI_PU_X1_17;


                        
                      
END_ACTION

ACTION IOHandleOutputs_Action:
                        ;
DEV_DSC_BUZZER := BUZZER_CONTROL;

                        
                      
END_ACTION

ACTION Main_Application_Action:
                        (* Call user application *)
Main();
                        
                      
END_ACTION

ACTION Other_Action:
                        (*###########################################################*)
(*This block is created implicit. Don't add own code to here.*)
(*###########################################################*)


                        
                      
END_ACTION

ACTION Other_EpecOut_Action:
                        (* tag EPEC_OUT_OTHER *)


IF G_Common.ParHandler.o_ParamAreaLocked THEN
	G_Common.ParHandler.DisableChanges(i_DisableChanges := FALSE);
END_IF


                      
END_ACTION
END_PROGRAM

CONFIGURATION Device
  RESOURCE Application ON PLC
    VAR_GLOBAL CONSTANT  (* Code_Template_constants *)
      G_NVRAM_6107_CODE_TEMPLATE_TOTAL : DWORD := 507904;  (* [Total size of NVRAM reserved for code template (IEC area 496 kB)] *)
      G_NVRAM_6107_GLOBE_DATA_SIZE : DWORD := 1024;  (* [Size of the GlobE NVRAM reservation] *)
      G_NVRAM_6107_AZURE_DATA_SIZE : DWORD := 1024;  (* [Size of the Azure NVRAM reservation] *)
      G_NVRAM_6107_AZURE_DATA_OFFSET : DWORD := 490496;  (* [Offset of the Azure NVRAM area.] *)
      G_NVRAM_6107_GLOBE_DATA_OFFSET : DWORD := 491520;  (* [Offset of the GlobE NVRAM area.] *)
      G_NUMBER_OF_PARAMETERS_NETWORK1 : INT := 0;  (* [Number of parameters in network] *)
      G_NVRAM_6107_OD_PAR_IMAGE_SIZE : DWORD := 204800;  (* [Size of the OD parameter area reservation.] *)
      G_NVRAM_6107_EVENT_LOG_SIZE : DWORD := 102400;  (* [Size of the EventLog reservation.] *)
      G_NVRAM_6107_USER_DATA_SIZE : DWORD := 102400;  (* [Size of the user NVRAM reservation.] *)
      G_NVRAM_6107_OD_PARAM_OFFSET : DWORD := 0;  (* [Offset for OD parameter area.] *)
      G_NVRAM_6107_EVENTLOG_OFFSET : DWORD := 204800;  (* [Offset of the EventLog area.] *)
      G_NVRAM_6107_USER_DATA_OFFSET : DWORD := 307200;  (* [Offset of the user NVRAM area.] *)
      G_NVRAM_MACHINETYPE_OFFSET : DWORD := 409600;  (* [Offset of the machine type area.] *)
      G_PARAMHANDLERKEYWORD : DWORD := 16#2464842F;  (* [ Parameterhandler keyword] *)
      G_PARAM_BLOCK_MAX_SIZE : WORD := 1024;  (* [ Maximum size of one parameter handler block] *)
      G_NVRAM_MACHINETYPE_SIZE : DWORD := 0;  (* [Size of the machine type area reservation.] *)
    END_VAR
    VAR_GLOBAL  (* Code_Template_globals *)
      G_RESET_MODULE : BOOL := FALSE;  (* [Flag indicates if unit is wanted to reset after current application cycle. Reset actions can be varied between platforms.] *)
      G_HWDiagnostics : HWD_Measurements_68xx;  (* [Function block instance which is used for voltage and temperature monitoring.] *)
      G_AddAllAutoGenEventsToLog : BOOL := TRUE;  (* [Add all automatically generated events to log.] *)
      G_OffDelayForAutoGenEvents : WORD := 50;  (* [Off delay for automatically generated events.] *)
      G_OnDelayForAutoGenEvents : WORD := 100;  (* [On delay for automatically generated events.] *)
      G_AIOverCurrentProtection_X1_5 : EPEC_6000INT.AIOverCurrentProtection;
      G_AIOverCurrentProtectionEnable_X1_5 : BOOL := TRUE;
      G_AIOverCurrentProtection_X1_17 : EPEC_6000INT.AIOverCurrentProtection;
      G_AIOverCurrentProtectionEnable_X1_17 : BOOL := TRUE;
      G_SystemOk : BOOL := FALSE;
      G_TempCPUHighLimit : INT := 900;
      G_TempCPULowLimit : INT := -300;
      G_TempPCBHighLimit : INT := 900;
      G_TempPCBLowLimit : INT := -300;
      G_SupplyVoltageHighLimit : UINT := 3000;
      G_SupplyVoltageLowLimit : UINT := 0;
      G_CycleTimeHighLimit : UINT := 50;
      G_Ref5VHighLimit : UINT := 550;
      G_Ref5VLowLimit : UINT := 450;
      G_AIBiasVoltageHighLimit : UINT := 780;
      G_AIBiasVoltageLowLimit : UINT := 680;
      G_RtcBackupVoltageLowLimit : UINT := 200;
      G_NVRAM_6107_StartAddress : DWORD;  (* [Pointer to the start of the NVRAM area.] *)
      G_NVRAM_6107_ODParamPointer : DWORD;  (* [Pointer to the start of the OD parameter image.] *)
      G_NVRAM_6107_EventLogPointer : DWORD;  (* [Pointer to the start of the EventLog] *)
      G_NVRAM_6107_UserDataPointer : DWORD;  (* [Pointer to the start of the user NVRAM area.] *)
      G_NVRAM_6107_GlobEDataPointer : DWORD;  (* [Pointer to the start of the GlobE NVRAM area.] *)
      G_NVRAM_6107_AzureDataPointer : DWORD;  (* [Pointer to the start of the Azure NVRAM area.] *)
      G_NVRAM_6107_J1939DM2LogPointer : DWORD;  (* [Pointer to the start of the J1939 DM2 NVRAM area.] *)
      G_NVRAM_MachineTypePointer : DWORD;  (* [Pointer to the start of the Machine type NVRAM area.] *)
      G_InitEntryReady : BOOL := FALSE;  (* [Init Flags] *)
      G_InitFlashReady : BOOL := FALSE;
      G_InitIOReady : BOOL := FALSE;
      G_InitBusReady : BOOL := FALSE;
      G_InitProtocolsCan1Ready : BOOL := FALSE;
      G_InitProtocolsCan2Ready : BOOL := FALSE;
      G_InitEventsReady : BOOL := FALSE;
      G_InitExitReady : BOOL := FALSE;
      G_ActiveError : BOOL := FALSE;
      G_MRAM_Shm : SystemSharedMemRegion;  (* [Shared memory structure which is used to get pointer to MRAM area for parameter saving.] *)
      G_CommsParamCounterSaveCmdOld : WORD := 0;  (* [Counter used to detect if communication parameters need to be saved] *)
      G_CommsParamCounterRestoreCmdOld : WORD := 0;  (* [Counter used to detect if communication parameters need to be restored] *)
      G_NodeIds : ARRAY[1..2] OF INT := [2, 2];
      G_CAN1_Channel : EPEC_6000CANVXD.Channel;
      G_InitProtocolsCan1State : InitCanProtocolStates := INIT_CANOPEN_PROTOCOLS;
      G_InitCANopenCan1Error : BOOL := FALSE;
      G_CANopenCan1ProtocolError : BOOL := FALSE;
      G_CAN2_Channel : EPEC_6000CANVXD.Channel;
      G_InitProtocolsCan2State : InitCanProtocolStates := INIT_CANOPEN_PROTOCOLS;
      G_InitCANopenCan2Error : BOOL := FALSE;
      G_CANopenCan2ProtocolError : BOOL := FALSE;
      G_NETWORK1_Parameters_CSVData : ARRAY[1..G_NUMBER_OF_PARAMETERS_NETWORK1] OF EPEC_PAR.CSVData;  (* [Parameter CSV configuration parameters] *)
      G_NETWORK1_Parameters_CsvFile : STRING(79) := 'Parameters_NETWORK1.csv';  (* [CSV file path and name] *)
      G_NETWORK1_Parameters_Count : INT;  (* [CSV File parameter count] *)
      G_NETWORK1_Parameters_ErrorCode : EPEC_PAR.CSVError;  (* [CSV error code] *)
      G_NETWORK1_Parameters_ErrorInLine : INT;  (* [Number of CSV line containing error] *)
      G_UserFolderPath : STRING(255);
    END_VAR
    VAR_GLOBAL  (* UserMramVariables *)
      G_pUserMramStructure : POINTER TO UserMramStructure;  (* [Pointer to the start of the NVRAM area.] *)
      G_UserMramStructureDefault : UserMramStructure;  (* [Pointer to the start of the OD parameter image.] *)
    END_VAR
    VAR_GLOBAL  (* IO *)
      AI_PU_X1_5 : WORD := 0;  (* [Pin 1.5 - lang.IO.FilteredAiValue] *)
      AI_X1_5 : WORD := 0;  (* [Pin 1.5 - lang.IO.FilteredAiValue] *)
      KL15_X1_6 : BOOL := FALSE;  (* [Pin 1.6 - KL15] *)
      AI_PU_X1_17 : WORD := 0;  (* [Pin 1.17 - lang.IO.FilteredAiValue] *)
      AI_X1_17 : WORD := 0;  (* [Pin 1.17 - lang.IO.FilteredAiValue] *)
    END_VAR
    VAR_GLOBAL  (* IO_INTERNAL *)
      TEMP_PCB : INT := 0;  (* Scaled PCB temperature [0.1 C] *)
      TEMP_CPU : INT := 0;  (* Scaled CPU temperature [0.1 C] *)
      SUPPLY_Volt : WORD := 0;  (* Scaled supply voltage [0.01 V] *)
      AIBias_Volt : WORD := 0;  (* Scaled AI bias voltage *)
      RTCBackup_Volt : WORD := 0;  (* Scaled RTC backup voltage *)
      Voltage12V : WORD := 0;  (* Scaled 12V voltage *)
      REF_5V : WORD := 0;  (* Scaled Ref 5 V voltage [10 mV]. *)
      REF_OUT_5V_Enable : BOOL := FALSE;  (* Enable for 5 V reference. *)
      REF_OUT_5V_OK : BOOL := FALSE;  (* 5 V refrence failure *)
      BUZZER_CONTROL : BOOL := FALSE;  (* Enable buzzer output control *)
      ALS_Volt : WORD := 0;  (* Unscaled ALS voltage measurement *)
    END_VAR
    VAR_GLOBAL  (* IO_CONFIG *)
      AI_SET_PU_X1_5 : BOOL := TRUE;  (* [Pin 1.5 - lang.IO.PullUpEnableSelectionForPin] *)
      AI_SET_mA_X1_5 : BOOL := FALSE;  (* [Pin 1.5 - lang.IO.ModeSelection] *)
      AI_SET_PU_X1_17 : BOOL := TRUE;  (* [Pin 1.17 - lang.IO.PullUpEnableSelectionForPin] *)
      AI_SET_mA_X1_17 : BOOL := FALSE;  (* [Pin 1.17 - lang.IO.ModeSelection] *)
    END_VAR
    {attribute 'qualified_only'}
    {attribute 'location' := '16#800'}
    {attribute 'analysis' := '-5, -6, -33, -43, -48'}
    VAR_GLOBAL  (* G_CAN1_VAR - NOTE! NOTE! NOTE! NOTE! NOTE! NOTE! NOTE! NOTE! NOTE! NOTE! NOTE! This object is created by Epec MultiTool User changes are overwritten when project is imported Content - CANopen OD index data *)
      DeviceType_Device1 : UDINT := 405;  (* [ 16#1000 Information about the device type] *)
      ErrorReg_Device1 : USINT := 0;  (* [ 16#1001 Error information] *)
      CAN1_TPDO_DUMMY : BYTE := 0;  (* [ 16#2128 PDO Dummy Variable Index] *)
      CAN1_RPDO_DUMMY : BYTE := 0;  (* [ 16#2129 PDO Dummy Variable Index] *)
      Parameter_CSV_unique_ID1 : UINT := 16#0000;  (* [ 16#2131 Parameter CSV unique ID] *)
      NonSafetyParameterAuthenticationStatus : BYTE := 0;  (* [ 16#21EE Authentication status for non-safety parameter editing] *)
      NonSafetyParameterPassword : STRING(79) := '';  (* [ 16#21EF Non-safety parameter password] *)
    END_VAR
    {attribute 'qualified_only'}
    {attribute 'location' := '16#800'}
    {attribute 'analysis' := '-5, -33, -43, -48'}
    VAR_GLOBAL  (* G_CAN1_RPDO - NOTE! NOTE! NOTE! NOTE! NOTE! NOTE! NOTE! NOTE! NOTE! NOTE! NOTE! This object is created by Epec MultiTool User changes are overwritten when project is imported Content - CAN1 mapped RPDO variables By all variable types, CAN in and out variables shall be at consecutive memory addresses, since they are mapped consecutively to same mapping OD index. G_CAN1_TPDO.TxPDOByte1 AT %MBx // PDO G_CAN1_TPDO.TxPDOByte<n> AT %MB<x+n> G_CAN1_RPDO.RxPDOByte1 AT %MB<x+n+1> Note! PDO, SRDO plain and SRDO inverted data is mapped to separate OD indexes. This means that it is NOT mandatory that they are in consecutive memory addresses. *)
      RAU_GPS_altitude AT %MB0 : REAL := 0;  (* [ ] *)
      RAU_GPS_latitude AT %MB4 : REAL := 0;  (* [ ] *)
      RAU_GPS_longitude AT %MB8 : REAL := 0;  (* [ ] *)
      RAU_GPS_NoOfSatellites AT %MB12 : REAL := 0;  (* [ ] *)
      RAU_GPS_quality AT %MB16 : REAL := 0;  (* [ ] *)
      RAU_GPS_speed AT %MB20 : REAL := 0;  (* [ ] *)
      RAU_GPS_error AT %MB32 : DWORD := 0;  (* [ ] *)
      RAU_Bits AT %MB37 : CAN1_RPDO_RAU_Bits;  (* [] *)
    END_VAR
    {attribute 'qualified_only'}
    {attribute 'location' := '16#800'}
    {attribute 'analysis' := '-5, -33, -43, -48'}
    VAR_GLOBAL  (* G_CAN1_TPDO - NOTE! NOTE! NOTE! NOTE! NOTE! NOTE! NOTE! NOTE! NOTE! NOTE! NOTE! This object is created by Epec MultiTool User changes are overwritten when project is imported Content - CAN1 mapped TPDO variables By all variable types, CAN in and out variables shall be at consecutive memory addresses, since they are mapped consecutively to same mapping OD index. G_CAN1_TPDO.TxPDOByte1 AT %MBx // PDO G_CAN1_TPDO.TxPDOByte<n> AT %MB<x+n> G_CAN1_RPDO.RxPDOByte1 AT %MB<x+n+1> Note! PDO, SRDO plain and SRDO inverted data is mapped to separate OD indexes. This means that it is NOT mandatory that they are in consecutive memory addresses. *)
      PT100 AT %MB24 : DWORD := 0;  (* [ ] *)
      PT1000 AT %MB28 : DWORD := 0;  (* [ ] *)
      Bits AT %MB36 : CAN1_TPDO_Bits;  (* [] *)
    END_VAR
    {attribute 'qualified_only'}
    {attribute 'global_init_slot' := '49991'}
    VAR_GLOBAL  (* G_CANopen_CAN1 - NOTE! NOTE! NOTE! NOTE! NOTE! NOTE! NOTE! NOTE! NOTE! NOTE! NOTE! This object is created by Epec MultiTool User changes are overwritten when project is imported Content - CANopen protocol variable definitions *)
      Device : EPEC_CANopen.Device;  (* [ CAN device] *)
      OD : EPEC_CANopen.OD;  (* [ Object Dictionary data] *)
      ODEntrys : ARRAY[1..89] OF EPEC_CANopen.ODEntry;  (* [] *)
      Protocols : ARRAY[1..6] OF EPEC_CANopen.ProtocolEntry;  (* [ Protocol data] *)
      HBCallbacks : ARRAY[1..1] OF EPEC_CANopen.CANopenHBCallback := [(i_NodeID := 1, i_Time := G_CANopen_CAN1_VAR.HBCTimes[1], i_pNext := 0)];  (* [ Heartbeat producer/consumer] *)
      HB : EPEC_CANopen.HBData;  (* [ Heartbeat producer/consumer protocol data] *)
      HB_Handler : EPEC_CANopen.CANopenHB;  (* [ Heartbeat producer/consumer protocol handler] *)
      MonitoredNodes : ARRAY[1..1] OF EPEC_CANopen.SlaveData := [(pHBCallback := ADR(HBCallbacks[1]), KeepAlive := TRUE, Reset := FALSE, Mandatory := TRUE, DisableStart := FALSE, QueryWithSDO := FALSE, ConfigurationDelay := 1000, SDOQueryInterval := 0, ConfigurationTimeout := 10)];  (* [ NMT] *)
      NMT : EPEC_CANopen.NMTData;  (* [ NMT protocol data] *)
      NMT_Handler : EPEC_CANopen.CANopenNMT;  (* [ NMT protocol handler] *)
      SSDO : EPEC_CANopen.SSDOData;  (* [ SDO server protocol data] *)
      SSDO_Handler : EPEC_CANopen.CANopenSDOServer;  (* [ SDO server protocol handler] *)
      PDO : EPEC_CANopen.PDOData;  (* [ PDO protocol data] *)
      PDOS : ARRAY[1..6] OF EPEC_CANopen.CANopenPDO;  (* [ PDO instances] *)
      PDO_Handler : EPEC_CANopen.CANopenPDOHandler;  (* [ PDO protocol handler] *)
      GFC : EPEC_CANopen.GFCData;  (* [ GFC protocol data] *)
      GFC_Handler : EPEC_CANopen.CANopenGFC;  (* [ GFC protocol handler] *)
      CSDOS : ARRAY[1..127] OF EPEC_CANopen.CANopenCSDO := [];  (* [ SDO client instances] *)
      SaveAll : EPEC_ODSave.SaveODSaveAll;  (* [] *)
      DeleteAll : EPEC_ODSave.SaveODDeleteAll;  (* [] *)
      SaveODHandler : EPEC_ODSave.SaveOD_Handler;  (* [] *)
      SaveData : ARRAY[0..3] OF EPEC_ODSave.SaveODSubIndexDescription := [(StartIndex := 16#1000, EndIndex := 16#FFFF, GroupNum := 1), (StartIndex := 16#1000, EndIndex := 16#1FFF, GroupNum := 1), (StartIndex := 16#2000, EndIndex := 16#FFFF, GroupNum := 1), (StartIndex := 16#0, EndIndex := 16#0, GroupNum := 1)];  (* [] *)
      SaveSubData1010h : EPEC_ODSave.SaveODSubService;  (* [] *)
      OD_ReOrg : EPEC_CANopen.CANopenODReOrg;  (* [] *)
    END_VAR
    {attribute 'qualified_only'}
    {attribute 'location' := '16#800'}
    {attribute 'global_init_slot' := '49990'}
    VAR_GLOBAL  (* G_CANopen_CAN1_VAR - NOTE! NOTE! NOTE! NOTE! NOTE! NOTE! NOTE! NOTE! NOTE! NOTE! NOTE! This object is created by Epec MultiTool User changes are overwritten when project is imported Content - *)
      OD_Error : EPEC_CANopen.Errors := EPEC_CANopen.Errors.NotInitialized;  (* [] *)
      ODSave_Error : EPEC_ODSave.SaveODErrors;  (* [] *)
      Callback_Error : EPEC_CANopen.Errors := EPEC_CANopen.Errors.NotInitialized;  (* [] *)
      ProtocolAdded : ARRAY[1..6] OF BOOL := [6(0)];  (* [] *)
      HBCTimes : ARRAY[1..1] OF UDINT := [UDINT#400];  (* [] *)
      HB_Error : EPEC_CANopen.Errors := EPEC_CANopen.Errors.NotInitialized;  (* [] *)
      NMT_Error : EPEC_CANopen.Errors := EPEC_CANopen.Errors.NotInitialized;  (* [] *)
      SSDO_Error : EPEC_CANopen.Errors := EPEC_CANopen.Errors.NotInitialized;  (* [] *)
      PDO_Error : EPEC_CANopen.Errors := EPEC_CANopen.Errors.NotInitialized;  (* [] *)
      GFC_Error : EPEC_CANopen.Errors := EPEC_CANopen.Errors.NotInitialized;  (* [] *)
      GFC_Status : BYTE;  (* [ GFC status] *)
      CSDO_Error : EPEC_CANopen.Errors := EPEC_CANopen.Errors.NotInitialized;  (* [] *)
      OD_REORG_Error : EPEC_CANopen.Errors := EPEC_CANopen.Errors.NotInitialized;  (* [] *)
      OdReOrgReady : BOOL := FALSE;  (* [ OD Reorganize operation ready] *)
      ODSave_OperationReady : BOOL := FALSE;  (* [] *)
      ODParametersInitialized : BOOL := FALSE;  (* [] *)
      SaveSigns1010 : ARRAY[0..3] OF DWORD;  (* [] *)
      InitProtocolsCanState : InitCanProtocolStates := InitCanProtocolStates.INIT_CANOPEN_PROTOCOLS;  (* [] *)
    END_VAR
    {attribute 'qualified_only'}
    {attribute 'location' := '16#800'}
    {attribute 'analysis' := '-43'}
    VAR_GLOBAL  (* G_CANopen_CAN1_Mappings - NOTE! NOTE! NOTE! NOTE! NOTE! NOTE! NOTE! NOTE! NOTE! NOTE! NOTE! This object is created by Epec MultiTool User changes are overwritten when project is imported Content - CAN1 mapped PDO and SRDO mapping variables *)
      PDO1_Mappings : ARRAY[1..G_CANOPEN_NUMBER_OF_LAST_PDO_MAP] OF DWORD := [DWORD#16#5FFF0108, 7(DWORD#16#0)];  (* [ PDO1 mappings G_CAN1_TPDO.Bits 8-1 = 7] *)
      PDO2_Mappings : ARRAY[1..G_CANOPEN_NUMBER_OF_LAST_PDO_MAP] OF DWORD := [DWORD#16#5FD70120, DWORD#16#5FD70220, 6(DWORD#16#0)];  (* [ PDO2 mappings G_CAN1_TPDO.PT100 G_CAN1_TPDO.PT1000 8-2 = 6] *)
      PDO3_Mappings : ARRAY[1..G_CANOPEN_NUMBER_OF_LAST_PDO_MAP] OF DWORD := [DWORD#16#5FFF0208, DWORD#16#5FD70320, 6(DWORD#16#0)];  (* [ PDO3 mappings G_CAN1_RPDO.RAU_Bits G_CAN1_RPDO.RAU_GPS_error 8-2 = 6] *)
      PDO4_Mappings : ARRAY[1..G_CANOPEN_NUMBER_OF_LAST_PDO_MAP] OF DWORD := [DWORD#16#5FB70120, DWORD#16#5FB70220, 6(DWORD#16#0)];  (* [ PDO4 mappings G_CAN1_RPDO.RAU_GPS_altitude G_CAN1_RPDO.RAU_GPS_latitude 8-2 = 6] *)
      PDO5_Mappings : ARRAY[1..G_CANOPEN_NUMBER_OF_LAST_PDO_MAP] OF DWORD := [DWORD#16#5FB70320, DWORD#16#5FB70420, 6(DWORD#16#0)];  (* [ PDO5 mappings G_CAN1_RPDO.RAU_GPS_longitude G_CAN1_RPDO.RAU_GPS_NoOfSatellites 8-2 = 6] *)
      PDO6_Mappings : ARRAY[1..G_CANOPEN_NUMBER_OF_LAST_PDO_MAP] OF DWORD := [DWORD#16#5FB70520, DWORD#16#5FB70620, 6(DWORD#16#0)];  (* [ PDO6 mappings G_CAN1_RPDO.RAU_GPS_quality G_CAN1_RPDO.RAU_GPS_speed 8-2 = 6] *)
    END_VAR
    TASK PLC_PRG_TASK(INTERVAL := T#10ms, PRIORITY := 1);
    PROGRAM PLC_PRG WITH PLC_PRG_TASK : PLC_PRG;
  END_RESOURCE
END_CONFIGURATION
